Fanuc KAREL source: kf00100.KL

-- PROVISIONAL review KL for V1013-1; original PC SHA256 b93eea018fdb6340290453f6600d5cfb3f03b7e170da46b28f126afa22a2944f
-- Incomplete behavior may be omitted. Consult companion uncertainty JSON. Do not deploy.
PROGRAM KF00100
%NOLOCKGROUP
BEGIN
  -- UNRESOLVED_PC offsets 5-16; opcodes 2E,23
  -- UNRESOLVED_PC offsets 21-32; opcodes 2E,23
  -- UNRESOLVED_PC offsets 37-63; opcodes 27,27,9D,22,1C,22,27,9D,31
  -- UNRESOLVED_PC offsets 68-72; opcodes 7F
END KF00100
